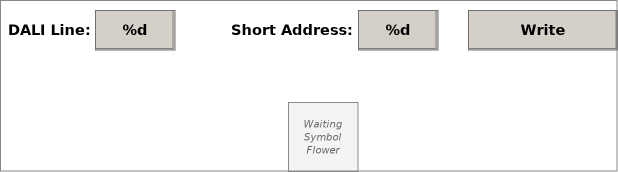
VISUALIZATION Visu_Part103Identify  // 618x172
    Button (468,10 150x40), "Write"
        OnMouseClick: execute { DALI_Commissioning.fbPart103IdentifyDevice.bWrite := TRUE; }
    WaitingSymbolFlower (288,102 70x70), invisible if: DALI_Commissioning.fbPart103MemoryPages.bHideWaitSymbol
    Textfield (228,10 130x40), "Short Address:"
    Button (358,10 80x40), "%d", text variable: DALI_Commissioning.fbPart103IdentifyDevice.nAddress
        OnMouseClick: write the text variable via Default, min 0, max 63, title "Insert Short Address"
    Group (5,10 170x40)
        Textfield (0,0 110x40), "DALI Line:"
        Button (90,0 80x40), "%d", text variable: GVL_Internal.nDALILine
            OnMouseClick: write the text variable via Default, min 1, max 10, title "Choose line"
END_VISUALIZATION

(* stored: Version 1.1.0.1
   Visu Visu_Part103Identify: Id {20e81529-1e04-4ad7-8b53-d10034b85d55} *)
